SUBAPPLICATION Uebung_009_AUDI (* Ticker (AX-Adapter basiert) *)
  (* Standard: 61499-2; Description: Copyright (c) 2023 Meisterschulen am Ostbahnhof This program and the accompanying materials are made available under the terms of the Eclipse Public License 2.0 which is available at https://www.eclipse.org/legal/epl-2.0/ SPDX-License-Identifier: EPL-2.0 *)
  (* Version 1.0, 2026-01-17, Franz Höpfinger, Meisterschulen am Ostbahnhof, initial API and implementation and/or initial documentation *)
  PACKAGE Uebungen;
  IMPORT Uebungen::const::UT::DefaultPool::OutputNumber_N1;
  IMPORT logiBUS::io::DQ::logiBUS_DO::Output_Q1;
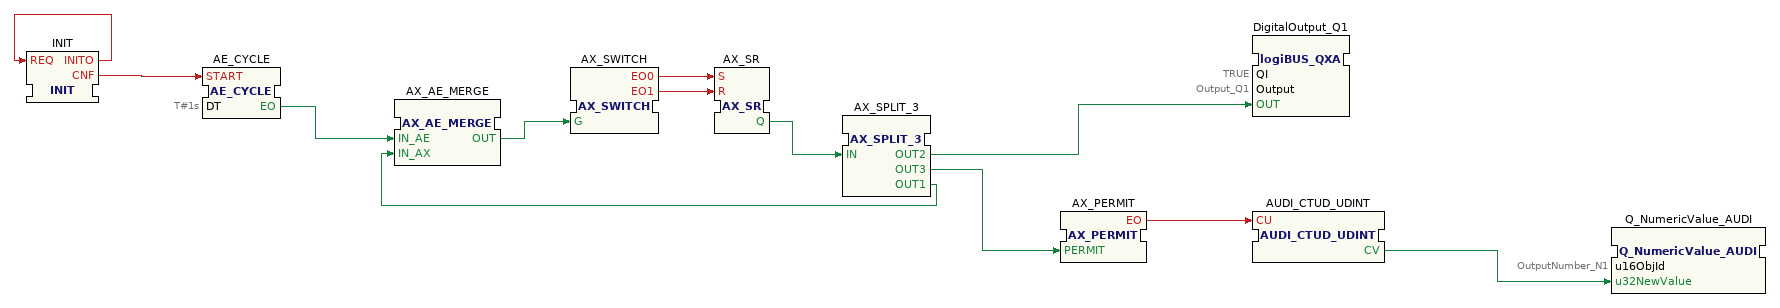
  FBS
    DigitalOutput_Q1 : logiBUS::io::DQ::logiBUS_QXA(QI := TRUE, Output := Output_Q1);
    AE_CYCLE : adapter::events::unidirectional::timers::AE_CYCLE(DT := T#1s);
    AX_SWITCH : adapter::events::unidirectional::AX_SWITCH;
    AX_SR : adapter::events::unidirectional::AX_SR;
    AX_PERMIT : adapter::events::unidirectional::AX_PERMIT;
    AUDI_CTUD_UDINT : adapter::events::unidirectional::AUDI_CTUD_UDINT;
    Q_NumericValue_AUDI : isobus::UT::Q::Q_NumericValue_AUDI(u16ObjId := OutputNumber_N1);
    AX_SPLIT_3 : adapter::events::unidirectional::AX_SPLIT_3;
    AX_AE_MERGE : adapter::events::unidirectional::AX_AE_MERGE;
    INIT : iec61131::bitwiseOperators::INIT;
  END_FBS
  EVENT_CONNECTIONS
    AX_SWITCH.EO0 TO AX_SR.S;
    AX_SWITCH.EO1 TO AX_SR.R;
    AX_PERMIT.EO TO AUDI_CTUD_UDINT.CU;
    INIT.INITO TO INIT.REQ;
    INIT.CNF TO AE_CYCLE.START;
  END_CONNECTIONS
  ADAPTER_CONNECTIONS
    AX_SPLIT_3.OUT2 TO DigitalOutput_Q1.OUT;
    AX_SR.Q TO AX_SPLIT_3.IN;
    AX_SPLIT_3.OUT3 TO AX_PERMIT.PERMIT;
    AUDI_CTUD_UDINT.CV TO Q_NumericValue_AUDI.u32NewValue;
    AX_AE_MERGE.OUT TO AX_SWITCH.G;
    AE_CYCLE.EO TO AX_AE_MERGE.IN_AE;
    AX_SPLIT_3.OUT1 TO AX_AE_MERGE.IN_AX;
  END_CONNECTIONS
END_SUBAPPLICATION
